// TIA Portal V15.1 export
// export: Created 2019-08-08T13:49:45.9546209Z, ExportSetting None, DisplayName Totally Integrated Automation Portal, DisplayVersion V15.1, DisplayName TIA Portal Openness, DisplayVersion V15.1, DisplayName STEP 7 Professional, DisplayVersion V15.1, DisplayName STEP 7 Safety, DisplayVersion V15.1, DisplayName WinCC Advanced, DisplayVersion V15.1
TYPE "UA_Method_Handle"
   STRUCT
      Pre : Struct   // PreCall Parameter
         Done : Bool;
         Busy : Bool;
         Error : Bool;
         Status : DWord;
      END_STRUCT;
      Post : Struct   // PostCall Parameter
         Done : Bool;
         Busy : Bool;
         Error : Bool;
         Status : DWord;
      END_STRUCT;
      Started : Bool;   // true=MethodCall started (pre done)
      Finished : Bool;   // true=MethodCall ended
      Result : DWord;   // Result of the Method Call
      Called : Bool;   // true=MethodeCall is called
      ErrorMessage : WString;   // Erroro Message
   END_STRUCT;
END_TYPE
